INTERFACE I_MetadataVisitor

METHOD VisitMetadatum
VAR_INPUT
	VisitingMetadatum : I_Metadata;
END_VAR
END_METHOD

END_INTERFACE

(* stored: Version 1.1.0.1, ProductVersion 3.1.4024.12
   Itf I_MetadataVisitor: Id {7671c5ec-d31c-0497-2f3e-d1fe1fbf32a2}
   Method VisitMetadatum: Id {74de62b9-0479-0783-29d3-341237058f5d} *)
